{attribute 'GeneratedUsingTerminal: EP9128-0021-0018'}
{attribute addProperty BoxType "EP9128-0021-0018"}
{attribute addProperty Id "A_0013_EP9128_0021_0019A_0013_EP9128_0021_0019_A3D9CE26523A_0010_EP9128_0021_0018_2_EP9128_1021EP9128_1FC0878B2A_0010_EP9128_0021_0018_3_EP9128_2021EP9128_1FC0878B2"}
{attribute addProperty CRC "2235624503"}
{attribute addProperty Size "527"}
TYPE A_0010_EP9128_0021_0018_8540EC37 EXTENDS EP9128_1FC0878B :
STRUCT
	{attribute addProperty Name "A_0013_EP9128_0021_0019"}
	{attribute addProperty PreviousPort "A_0010(EP9128-0021-0018) : D"}
	A_0013_EP9128_0021_0019 : A_0013_EP9128_0021_0019_A3D9CE26;
	{attribute addProperty Name "A_0010_EP9128_0021_0018_2_EP9128_1021"}
	{attribute addProperty PreviousPort "A_0010(EP9128-0021-0018) : C"}
	A_0010_EP9128_0021_0018_2_EP9128_1021 : EP9128_1FC0878B;
	{attribute addProperty Name "A_0010_EP9128_0021_0018_3_EP9128_2021"}
	{attribute addProperty PreviousPort "A_0010(EP9128-0021-0018)_2 (EP9128-1021) : C"}
	A_0010_EP9128_0021_0018_3_EP9128_2021 : EP9128_1FC0878B;
END_STRUCT
END_TYPE

(* stored: Version 1.2.0.0, ProductVersion 3.1.4024.9
   DUT A_0010_EP9128_0021_0018_8540EC37: Id {347ee968-9f03-4148-a404-6dcc33e08d2f} *)
